// TIA Portal V17 export
// export: Created 2023-04-03T06:31:41.4394818Z, ExportSetting WithDefaults, DisplayName Totally Integrated Automation Portal, DisplayVersion V17 Update 4, DisplayName TIA Portal Openness, DisplayVersion V17 Update 4, DisplayName TIA Portal Version Control Interface, DisplayVersion V17, DisplayName STEP 7 Professional, DisplayVersion V17 Update 4, DisplayName STEP 7 Safety, DisplayVersion V17, DisplayName WinCC Professional, DisplayVersion V17 Update 4
VAR_GLOBAL   // PLC tag table "Remote profinet Pems"
   "Emergency push button PEMS" AT %I50.0 : Bool;   // Slot01_In_00_513S1
   Available AT %I50.4 : Bool;   // Slot01_In_04_AVAILABLE
   "Emergency stop feeback contactors" AT %I50.1 : Bool;   // Slot01_In_01_517K1
   "Fire detection system Extinguisher activation" AT %I50.5 : Bool;   // Slot01_In_05_081K3
   "Push button emergncy reset" AT %I50.2 : Bool;   // Slot01_In_02_513P1
   "Spare(15)" AT %I50.6 : Bool;   // Slot01_In_06_SPARE
   "Spare(16)" AT %I50.3 : Bool;   // Slot01_In_03_SPARE
   "Spare(17)" AT %I50.7 : Bool;   // Slot01_In_07_SPARE
   "E - stop from PCS1" AT %I51.0 : Bool;   // Slot02_In_00_PCS1
   "E - stop from PCS2" AT %I51.4 : Bool;   // Slot02_In_04_PCS2
   "E - stop from external" AT %I51.1 : Bool;   // Slot02_In_01_EXTERNAL
   "Spare(18)" AT %I51.5 : Bool;   // Slot02_In_05_SPARE
   "Spare(19)" AT %I51.2 : Bool;   // Slot02_In_02_SPARE
   "CMV signal PCS1" AT %I51.6 : Bool;   // Slot02_In_06
   "CMV signal PCS2" AT %I51.3 : Bool;   // Slot02_In_03
   "Spare(20)" AT %I51.7 : Bool;   // Slot02_In_07_SPARE
   "Spare(22)" AT %I10.0 : Bool;   // Slot04_In_00_519K1
   "Spare(23)" AT %I10.1 : Bool;   // Slot04_In_04_519K2
   "Spare(24)" AT %I10.2 : Bool;   // Slot04_In_01_519K3
   "Spare(25)" AT %I10.3 : Bool;   // Slot04_In_05_519K4
   "Available(1)" AT %I10.4 : Bool;   // Slot04_In_02_AVAILABLE
   "Available(2)" AT %I10.5 : Bool;   // Slot04_In_06_AVAILABLE
   "Spare(26)" AT %I10.6 : Bool;   // Slot04_In_03_SPARE
   "Spare(27)" AT %I10.7 : Bool;   // Slot04_In_07_SPARE
   "Surge suppressor" AT %I11.0 : Bool;   // Slot05_In_00_01F1
   "Main circuit breaker(1)" AT %I11.1 : Bool;   // Slot05_In_04_3Q1
   "Pw supply Hvac CATL RH" AT %I11.2 : Bool;   // Slot05_In_01_11F1
   "Pw supply Hvac CATL LH" AT %I11.3 : Bool;   // Slot05_In_05_17F1
   "Pw supply Hvac PEMS" AT %I11.4 : Bool;   // Slot05_In_02_23Q1
   "Pw supply SPARE" AT %I11.5 : Bool;   // Slot05_In_06_25F1
   "Pw supply SPARE(1)" AT %I11.6 : Bool;   // Slot05_In_03_25F2
   "Pw supply Fire detection board" AT %I11.7 : Bool;   // Slot05_In_07_25F3
   "Signal Hvac Outdoor" AT %I12.0 : Bool;   // Slot06_In_00
   "Pw supply incoming line UPS" AT %I12.1 : Bool;   // Slot06_In_04_25F4
   "General breaker output of UPS" AT %I12.2 : Bool;   // Slot06_In_01_103F1
   "Pw supply control CATL RH (1RH - 12RH)" AT %I12.3 : Bool;   // Slot06_In_05_105F1
   "Pw supply control CATL LH (1LH - 12LH)" AT %I12.4 : Bool;   // Slot06_In_02_107F1
   "Pw supply Unit 1 230Vac/24Vdc" AT %I12.5 : Bool;   // Slot06_In_06_109F2
   "Pw supply Unit 2 230Vac/24Vdc" AT %I12.6 : Bool;   // Slot06_In_03_109F3
   "Pw supply shunt opening release" AT %I12.7 : Bool;   // Slot06_In_07_111F1
   "Pw supply spare(2)" AT %I13.0 : Bool;   // Slot07_In_00_111F2
   "Pw supply 24Vdc Comm equipment" AT %I13.1 : Bool;   // Slot07_In_04
   "Pw supply 24Vdc Safety PLC" AT %I13.2 : Bool;   // Slot07_In_01
   "Pw supply 24Vdc Digital PLC" AT %I13.3 : Bool;   // Slot07_In_05
   "Pw supply 24Vdc Available" AT %I13.4 : Bool;   // Slot07_In_02
   "Pw supply 24Vdc I/O internal PLC" AT %I13.5 : Bool;   // Slot07_In_06
   "Pw supply 24Vdc I/O external PLC" AT %I13.6 : Bool;   // Slot07_In_03
   "Pw supply 24Vdc Fire detection system" AT %I13.7 : Bool;   // Slot07_In_07
   "Pw supply 24Vdc CATL RH (MBMU - ETH)" AT %I14.0 : Bool;   // Slot08_In_00
   "Pw supply 24Vdc CATL LH (MBMU - ETH)" AT %I14.1 : Bool;   // Slot08_In_04
   "Pw supply 24Vdc DO safety to PCS" AT %I14.2 : Bool;   // Slot08_In_01
   "Available(3)" AT %I14.3 : Bool;   // Slot08_In_05
   "Available(4)" AT %I14.4 : Bool;   // Slot08_In_02
   "Available(5)" AT %I14.5 : Bool;   // Slot08_In_06
   "Available(6)" AT %I14.6 : Bool;   // Slot08_In_03
   "Available(7)" AT %I14.7 : Bool;   // Slot08_In_07
   "Pw supply Spare(3)" AT %I15.0 : Bool;   // Slot09_In_00_111F3
   "Available(8)" AT %I15.1 : Bool;   // Slot09_In_04
   "Available(9)" AT %I15.2 : Bool;   // Slot09_In_01
   "Available(10)" AT %I15.3 : Bool;   // Slot09_In_05
   "Available(11)" AT %I15.4 : Bool;   // Slot09_In_02
   "Fire detection system PRE-ALARM" AT %I15.5 : Bool;   // Slot09_In_06_81K1
   "Fire detection system FAULT" AT %I15.6 : Bool;   // Slot09_In_03_81K2
   "Fire detection system SPARE" AT %I15.7 : Bool;   // Slot09_In_07_81K4
   "Treshold 40°C thermostat" AT %I16.0 : Bool;   // Slot10_In_00_531S1
   "Treshold 55°C thermostat" AT %I16.1 : Bool;   // Slot10_In_04_531S2
   "Spare(28)" AT %I16.2 : Bool;   // Slot10_In_01
   "Pems panel open 1" AT %I16.3 : Bool;   // Slot10_In_05_531S4
   "Pems panel open 2" AT %I16.4 : Bool;   // Slot10_In_02_531S5
   "Spare(29)" AT %I16.5 : Bool;   // Slot10_In_06
   "Spare(30)" AT %I16.6 : Bool;   // Slot10_In_03
   "Spare(31)" AT %I16.7 : Bool;   // Slot10_In_07
   "Spare(32)" AT %I17.0 : Bool;   // Slot11_In_00
   "Spare(33)" AT %I17.1 : Bool;   // Slot11_In_04
   "Spare(34)" AT %I17.2 : Bool;   // Slot11_In_01
   "Spare(35)" AT %I17.3 : Bool;   // Slot11_In_05
   "Spare(36)" AT %I17.4 : Bool;   // Slot11_In_02
   "Spare(37)" AT %I17.5 : Bool;   // Slot11_In_06
   "Spare(38)" AT %I17.6 : Bool;   // Slot11_In_03
   "Spare(39)" AT %I17.7 : Bool;   // Slot11_In_07
   "Pw supply control CATL RH" AT %I18.0 : Bool;   // Slot12_In_00_551Q1
   "Pw supply control CATL LH" AT %I18.1 : Bool;   // Slot12_In_04_551Q2
   "Spare PCS1" AT %I18.2 : Bool;   // Slot12_In_01_551K1
   "Spare PCS2" AT %I18.3 : Bool;   // Slot12_In_05_551K2
   "UPS shut down any mode(1)" AT %I18.4 : Bool;   // Slot12_In_02_551K3
   "DC power ON battey bank closed RH" AT %I18.5 : Bool;   // Slot12_In_06_551K4
   "DC power ON battey bank closed LH" AT %I18.6 : Bool;   // Slot12_In_03_551K5
   "Spare(40)" AT %I18.7 : Bool;   // Slot12_In_07_551K6
   "Emergency stop General Breaker" AT %Q62.0 : Bool;   // xFDO_Slot03_Out01_517k1
   "Emergency stop UPS breaker" AT %Q62.1 : Bool;   // xFDO_Slot03_Out02_517k2
   "Emergency stop PCS1 (PE)" AT %Q62.2 : Bool;   // xFDO_Slot03_Out03_517k3
   "Emergency stop PCS2 (PE)" AT %Q62.3 : Bool;   // xFDO_Slot03_Out04_517k4
   "Emergency stop RESET shunt opening release" AT %Q62.4 : Bool;   // xFDO_Slot03_Out05_517k5
   spare AT %Q62.5 : Bool;   // xFDO_Slot03_Out06_517k6
   "Controls HVAC" AT %Q62.6 : Bool;   // xFDO_Slot03_Out07_517k7
   "Light emergency reset" AT %Q62.7 : Bool;   // xFDO_Slot03_Out08_513P1
END_VAR
